{attribute 'qualified_only'}
{attribute 'strict'}
{attribute 'to_string'}
TYPE ST_EStationHandshake :
(	
	Load := 1,
	CameraCheck:=2,
	
);
END_TYPE

(* stored: Version 1.1.0.1
   DUT ST_EStationHandshake: Id {d9b2890f-80b2-4461-acaf-694e8b5b19bc} *)
